Staubli VAL3: encodeAck.pgx

public program encodeAck()
begin
  // Copyright (c) 2016, Ocado Technology - Robotics Research Team
  //
  // Licensed under the Apache License, Version 2.0 (the "License");
  // you may not use this file except in compliance with the License.
  // You may obtain a copy of the License at
  //
  //     http://www.apache.org/licenses/LICENSE-2.0
  //
  // Unless required by applicable law or agreed to in writing, software
  // distributed under the License is distributed on an "AS IS" BASIS,
  // WITHOUT WARRANTIES OR CONDITIONS OF ANY KIND, either express or implied.
  // See the License for the specific language governing permissions and
  // limitations under the License.



  switch rosGenericMsg.header.nMsgType
    case nStdMsgType["JOINT_TRAJ_PT"]
      call encTrajPtAck()
    break
    case nStdMsgType["JOINT_TRAJ_PT_FULL"]
      call encTrajPtFAck()
    break
    default
    break
  endSwitch
end
